// TIA Portal V19 export
VAR_GLOBAL   // PLC tag table "Default tag table"
   FirstScan AT %M101.0 : Bool;
   DiagStatusUpdate AT %M101.1 : Bool;
   AlwaysTRUE AT %M101.2 : Bool;
   AlwaysFALSE AT %M101.3 : Bool;
   SpeedAxis_1_Actor_Interface_AddressIn AT %I256.0 : "PD_TEL1_IN";
   SpeedAxis_1_Actor_Interface_AddressOut AT %Q256.0 : "PD_TEL1_OUT";
   POT2_Warning AT %M20.4 : Bool;
   System_Byte AT %MB101 : Byte;
   Clock_Byte AT %MB100 : Byte;
   Clock_10Hz AT %M100.0 : Bool;
   Clock_5Hz AT %M100.1 : Bool;
   "Clock_2.5Hz" AT %M100.2 : Bool;
   Clock_2Hz AT %M100.3 : Bool;
   "Clock_1.25Hz" AT %M100.4 : Bool;
   Clock_1Hz AT %M100.5 : Bool;
   "Clock_0.625Hz" AT %M100.6 : Bool;
   "Clock_0.5Hz" AT %M100.7 : Bool;
   ConveyorWorking AT %M6.0 : Bool;   // Conveyor Diagnostic Tag
   OS7 AT %M21.3 : Bool;
   PB_Green_from_1200 AT %I100.0 : Bool;
   PB_Blue_from_1200 AT %I100.1 : Bool;
   POT_from_1200 AT %IW102 : Word;
END_VAR
